// TIA Portal V20 export
TYPE "Log_Data_String20"
// stored: Namespace ProductionLine
   STRUCT
      DataType : Byte;
      Representation : Byte;
      RepreLength : Byte;
      Reserve : Byte;
      Data : String[20];
   END_STRUCT;
END_TYPE
